FUNCTION_BLOCK FB_TestApplicationConfigRoot EXTENDS FB_ApplicationConfigRoot
VAR_OUTPUT
	IoRegistrationCalls : UINT;
	BaseUnitRegistrationCalls : UINT;
	ModuleTypeRegistrationCalls : UINT;
	ModuleCycleCalls : UINT;
	RegistrationOrderValid : BOOL := TRUE;
END_VAR
VAR
	_nRegistrationStep : UINT;
END_VAR

METHOD PROTECTED H_RegisterBaseUnits
BaseUnitRegistrationCalls := BaseUnitRegistrationCalls + 1;
_nRegistrationStep := _nRegistrationStep + 1;
RegistrationOrderValid := RegistrationOrderValid AND (_nRegistrationStep = 2);
M_RegisterBaseUnit(BaseUnit := GVL_IO.NC_Axis1);
END_METHOD

METHOD PROTECTED H_RegisterIo
IoRegistrationCalls := IoRegistrationCalls + 1;
_nRegistrationStep := _nRegistrationStep + 1;
RegistrationOrderValid := RegistrationOrderValid AND (_nRegistrationStep = 1);
M_RegisterIoNode(
	Variable := GVL_IO.Term4_EL1889.Chl[1],
	Access := E_VariableAccess.ReadOnly);
END_METHOD

METHOD PROTECTED H_RegisterModuleTypes
ModuleTypeRegistrationCalls := ModuleTypeRegistrationCalls + 1;
_nRegistrationStep := _nRegistrationStep + 1;
RegistrationOrderValid := RegistrationOrderValid AND (_nRegistrationStep = 3);

// Deliberately fail the last registration stage so the test does not load a
// target-dependent JSON file and can verify first-error latching deterministically.
M_RegisterModuleType(
	ModuleTypeName := '',
	Adapter := 0);
END_METHOD

METHOD PROTECTED H_RunModules
VAR_INPUT
	VariableNodeReader : I_VariableNodeReader;
END_VAR
VAR_IN_OUT CONSTANT
	SystemContext : ST_SystemContext;
END_VAR
ModuleCycleCalls := ModuleCycleCalls + 1;
END_METHOD

METHOD PUBLIC M_InvokeRunModulesForTest
VAR_IN_OUT CONSTANT
	SystemContext : ST_SystemContext;
END_VAR
VAR
	VariableNodeReader : I_VariableNodeReader;
END_VAR
H_RunModules(
	SystemContext := SystemContext,
	VariableNodeReader := VariableNodeReader);
END_METHOD

END_FUNCTION_BLOCK

(* stored: Version 1.1.0.1, ProductVersion 3.1.4026.18
   POU FB_TestApplicationConfigRoot: Id {e4981d98-9134-4415-9992-6292c045e5c3}, SpecialFunc None
   Method H_RegisterBaseUnits: Id {3ca42fbd-31b2-4f1b-96bb-9c46e0435a54}
   Method H_RegisterIo: Id {065f8bf1-a169-4678-bca4-01b22ccc6b39}
   Method H_RegisterModuleTypes: Id {befe120e-3f23-4a08-abb5-2157056b9ffd}
   Method H_RunModules: Id {f9ad22a2-295d-4247-ab88-07e642fac0f1}
   Method M_InvokeRunModulesForTest: Id {5181f65c-80a1-4944-a6ce-121041357bdb} *)
